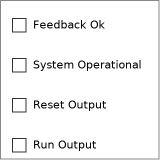
VISUALIZATION Vi_Sim_Safety  // 160x160
VAR_IN_OUT
	obj			: Safety;
END_VAR
    Checkbox (10,10 150x30), "Feedback Ok", variable: obj.bFeedbackOk
    Checkbox (10,50 150x30), "System Operational", variable: obj.bOperational
    Checkbox (10,90 150x30), "Reset Output", variable: obj.bReset
    Checkbox (10,130 150x30), "Run Output", variable: obj.bRun
END_VISUALIZATION

(* stored: Version 1.1.0.1
   Visu Vi_Sim_Safety: Id {24c1356e-8238-4fbe-9eed-9467c26d3bdd} *)
